(* IEC 61131-3 sources: iec/syntax/tests/data, 4 files *)

(* ---- struct_decl.st ---- *)
TYPE UDT_STRUCTANYPTR
    STRUCT
        S7Code : BYTE; // Code for S7 = 0x10
        DataType : BYTE; // Code for data type = 0x02 = byte
        Length : INT; // Repetition factor = Send/receive length
        DBNumber : INT; // Data block Number
        MemoryArea : BYTE; // Specified memory area = 0x84 = data block
        ByteAddressMSB : BYTE; // Byte address most significant bits
        ByteAddressLSB : WORD; // Byte address least significant bits
    END_STRUCT
END_TYPE

(* ---- id_function.st ---- *)
FUNCTION mqttGetNextMessageID : INT
BEGIN
    mqttData.nextMsgId := mqttData.nextMsgId + 1;

    IF (mqttData.nextMsgId <= 0) THEN
        mqttData.nextMsgId := 1;
    END_IF;

    mqttGetNextMessageID := mqttData.nextMsgId;
END_FUNCTION

(* ---- function_block.st ---- *)
FUNCTION_BLOCK mqttRuntime

VAR_INPUT
    IN      :   BOOL;
    RES     :   BOOL;
END_VAR

VAR_OUTPUT
    RTIME   :   TIME;
END_VAR

VAR
    last    :   DINT;
    now     :   DINT;
    run     :   DINT;
    FP_IN   :   BOOL;
END_VAR

BEGIN

IF IN AND NOT FP_IN THEN
    last := 0;
    FP_IN := true;
END_IF;

IF NOT IN AND FP_IN THEN
    FP_IN := false;
END_IF;

IF IN AND NOT RES THEN
    now := DWORD_TO_DINT(Unixtime());
    IF last = 0 THEN
        last := now;
    ELSE
        run := run + (now - last);
        last := now;
    END_IF;

END_IF;

IF IN AND RES THEN
    run := 0;
    now := 0;
    last := 0;
ELSIF NOT IN AND RES THEN
    run := 0;
    now := 0;
    last := 0;
END_IF;

IF run >= 2073600 THEN
    run := 0;
END_IF;

RTIME := DINT_TO_TIME(run * 1000);

END_FUNCTION_BLOCK

(* ---- hello_world.st ---- *)
PROGRAM MAIN
    VAR
        i: int;
        count: int;
    END_VAR

    for i := 0 TO 7 do
        count := count + i;
    end_for;

END_PROGRAM
